(* this fb for burner type that request off power and turn on again to reset it*)
FUNCTION_BLOCK FB_BurnerControlEcoFlamV3 EXTENDS FB_BurnerControlEcoFlamV2 IMPLEMENTS I_BurnerControlEcoFlamV3
VAR
	poOnOff : FB_DigitalOutput;
	poGasLv1 : FB_DigitalOutput;
	poGasLv2 : FB_DigitalOutput;
	eResetState : E_EcoFlamStateResetV3;
	tonDelayOffPower : TON;
	tonDelayOnPower : TON;
	timeDelayOnOffPower : TIME := T#2S;
END_VAR

IF IsRefActivePower THEN
	CASE ActivePowerType OF
		ACTIVE_POWER_TYPE_FEEDBACK:
			poOnOff.Out := ifActivePower.PowerOnIsCalled;
			poGasLv1.Out := ifActivePower.PowerOnIsCalled;
		ACTIVE_POWER_TYPE_NO_FEEDBACK:
			poOnOff.Out := ifActivePowerNoFB.PowerOnIsCalled;
			poGasLv1.Out := ifActivePowerNoFB.PowerOnIsCalled;
	END_CASE
END_IF
bError := piFault.In;
piFireSussess();
StateMachine();
tonMeasurementTimer(PT := tMeasurement);
IF piFireSussess.RisingTrigger AND eState=ECOFLAM_IGNITION THEN
	tBurnSuccess	:= 	tonMeasurementTimer.ET;				
END_IF

tonReset(
	in := (eState=ECOFLAM_RESET AND eResetState=ECOFLAM_V3_RESET_PORESET_ON),
	PT := timeReset
);
poReset();
poReset.Out := tonReset.IN;
tonDelayOffPower(
	IN := eState=ECOFLAM_RESET AND eresetstate=ECOFLAM_V3_RESET_TURN_OFF,
	PT := timeDelayOnOffPower
);
tonDelayOnPower(
	IN := eState=ECOFLAM_RESET AND eresetstate=ECOFLAM_V3_RESET_TURN_ON,
	PT := timeDelayOnOffPower
);

METHOD PROTECTED MS_Aborting
VAR_INPUT
END_VAR
SUPER^.MS_Aborting();
eResetState := ECOFLAM_V3_RESET_TURN_OFF;
END_METHOD

METHOD PROTECTED MS_Reset : BOOL
piFireSussess.MR_Reset();
bInit 		:= FALSE;
bAbort		:= FALSE;
bIgnition 	:= FALSE;
bStop 		:= FALSE;

CASE eResetState OF
	ECOFLAM_V3_RESET_TURN_OFF:
		CASE THIS^.eActivePowerType OF
			ACTIVE_POWER_TYPE_NO_FEEDBACK:
				ifActivePowerNoFB.MR_PowerOFF();
				IF tonDelayOffPower.Q THEN
					eResetState := ECOFLAM_V3_RESET_TURN_ON;
				END_IF
			ACTIVE_POWER_TYPE_FEEDBACK:
				ifActivePower.MR_PowerOFF();
				IF tonDelayOffPower.Q
					AND NOT ifActivePower.Powered AND NOT ifActivePower.Busy
				THEN
					eResetState := ECOFLAM_V3_RESET_TURN_ON;
				END_IF
		END_CASE
		
	ECOFLAM_V3_RESET_TURN_ON:
		CASE THIS^.eActivePowerType OF
			ACTIVE_POWER_TYPE_NO_FEEDBACK:
				ifActivePowerNoFB.MR_PowerON();
				IF tonDelayOnPower.Q THEN
					eResetState := ECOFLAM_V3_RESET_PORESET_ON;
				END_IF
			ACTIVE_POWER_TYPE_FEEDBACK:
				ifActivePower.MR_PowerON();
				IF (ifActivePower.Powered AND NOT ifActivePower.Busy)
					AND tonDelayOnPower.Q
				THEN
					eResetState := ECOFLAM_V3_RESET_PORESET_ON;
				END_IF
		END_CASE
		
	ECOFLAM_V3_RESET_PORESET_ON:
		IF tonReset.Q THEN
			eState := ECOFLAM_RESET_DONE;
		END_IF
END_CASE
END_METHOD

METHOD PROTECTED MS_ResetDone
VAR_INPUT
END_VAR
SUPER^.MS_ResetDone();
eResetState := ECOFLAM_V3_RESET_TURN_OFF;
END_METHOD

PROPERTY Ref_poGasLv1 : REFERENCE TO FB_DigitalOutput
GET
Ref_poGasLv1 ref= poGasLv1;
END_GET
END_PROPERTY

PROPERTY Ref_poGasLv2 : REFERENCE TO FB_DigitalOutput
GET
Ref_poGasLv2 ref= poGasLv2;
END_GET
END_PROPERTY

PROPERTY Ref_poOnOff : REFERENCE TO FB_DigitalOutput
GET
Ref_poOnOff ref= poOnOff;
END_GET
END_PROPERTY

END_FUNCTION_BLOCK

(* stored: Version 1.1.0.1, ProductVersion 3.1.4024.12
   POU FB_BurnerControlEcoFlamV3: Id {40ab636a-b8a1-4bda-af1e-6b0c6d112d1d}, SpecialFunc None
   Method MS_Aborting: Id {9ffa11ae-f174-4b02-a427-3b46217ea8c0}
   Method MS_Reset: Id {68651d15-8acf-45b4-9d27-be04aeff67a5}
   Method MS_ResetDone: Id {ed21c178-5293-4e51-a4fd-a92879738ada}
   Property Ref_poGasLv1: Id {4d9794b6-a63a-48e4-a338-0d5cc6f7d7a3}
   Get Get: Id {4082d1c2-5f6a-4c9f-858d-2b1e5100ee74}
   Property Ref_poGasLv2: Id {a4cde0dd-6c9e-4d2f-9a7c-c92a49365c5f}
   Get Get: Id {46d21bbb-9b87-4049-a477-f573fdec9b19}
   Property Ref_poOnOff: Id {e8e58ddd-0d8a-44f1-a09b-25662cbd80c9}
   Get Get: Id {142be0d3-406e-4b2d-9dbb-32069800c34a} *)
